// TIA Portal V20 export
DATA_BLOCK "BA040AZSCDR25_MendrelAnodeRearAxisYCamMain"   // DB285, Motion_DB
// stored: InstanceOfName TO_Cam_10k, OfSystemLibElement TO_Cam_10k, OfSystemLibVersion 9.0
TO_Cam_10k   // technology object, version 9.0
   // // inherited from TO_CamBase
   // // inherited from TO_Object
   // VAR
   //    InterpolationSettings { S7_SetPoint := 'True'} : TO_Cam_Struct_InterpolationSettings;
   //    StatusCam { ExternalWritable := 'False'; S7_SetPoint := 'True'} : TO_Cam_Struct_StatusCam;
   //    Point { S7_SetPoint := 'True'} : Array[1..10000] of TO_Cam_Struct_PointData;
   //    ValidPoint : Array[1..10000] of Bool;
   //    Segment { S7_SetPoint := 'True'} : Array[1..50] of TO_Cam_Struct_SegmentData;
   //    ValidSegment : Array[1..50] of Bool;
   //    StatusWord { ExternalWritable := 'False'} : DWord;
   //    ErrorWord { ExternalWritable := 'False'} : DWord;
   //    ErrorDetail { ExternalWritable := 'False'; S7_SetPoint := 'True'} : TO_Struct_ErrorDetail;
   //    WarningWord { ExternalWritable := 'False'} : DWord;
   // END_VAR
BEGIN
   InterpolationSettings.InterpolationMode := 1;
END_DATA_BLOCK
